// TwinCAT 3 PLC project StetigerPID_Regler
// ProgramVersion: 3.1.4022.1
// libraries:
//   Tc2_ControllerToolbox, * (Beckhoff Automation GmbH)
//   Tc2_Standard, * (Beckhoff Automation GmbH)
//   Tc2_System, * (Beckhoff Automation GmbH)
//   Tc2_TempController, * (Beckhoff Automation GmbH)
//   Tc2_Utilities, * (Beckhoff Automation GmbH)
//   Tc3_Module, * (Beckhoff Automation GmbH)
// project tree:
//   GVLs/ AN.TcGVL, DIO.TcGVL, dSub.TcGVL
//   / PlcTask.TcTTO
//   POUs/ MAIN.TcPOU, StetigerPID_Regler.TcPOU
// real-time tasks:
//   TASK PlcTask: cycle T#10ms, priority 20, ADS port 350
// motion (NC):
//   TASK NC-Task 1 SAF: cycle T#2ms, priority 4, ADS port 501
//   TASK NC-Task 1 SVB: cycle T#10ms, priority 8, ADS port 511
//   AXIS Axis 1 (id 1)
//     OtherSettings: AllowMotionCmdToSlave=true
//     encoder EncType=4
//       EncPara: MaxCount=#x0000ffff
//         Inc: RefSoftSyncMask=#x0000ffff
//     drive DrvType=24
//       Analog: ScaleFactorActTorque=0.1
//       TimeComp: TaskDelayCycles=1
//     controller CtrType=1
//       CtrPara: PriorControlFactor=1
//         Observer: BandWidth=20
//   AXIS Axis 2 (id 2)
//     OtherSettings: AllowMotionCmdToSlave=true
//     encoder EncType=4
//       EncPara: MaxCount=#x0000ffff
//         Inc: RefSoftSyncMask=#x0000ffff
//     drive DrvType=24
//       Analog: ScaleFactorActTorque=0.1
//       TimeComp: TaskDelayCycles=1
//     controller CtrType=1
//       CtrPara: PriorControlFactor=1
//         Observer: BandWidth=20
//   AXIS Axis 3 (id 3)
//     OtherSettings: AllowMotionCmdToSlave=true
//     encoder EncType=4
//       EncPara: MaxCount=#x0000ffff
//     drive DrvType=23
//       Analog: ScaleFactorActTorque=0.1
//       TimeComp: TaskDelayCycles=1
//     controller CtrType=1
//       CtrPara: PriorControlFactor=1
//         Observer: BandWidth=20
//   AXIS Axis 4 (id 4)
//     OtherSettings: AllowMotionCmdToSlave=true
//     encoder EncType=4
//       EncPara: MaxCount=#x0000ffff
//     drive DrvType=23
//       Analog: ScaleFactorActTorque=0.1
//       TimeComp: TaskDelayCycles=1
//     controller CtrType=1
//       CtrPara: PriorControlFactor=1
//         Observer: BandWidth=20
//   AXIS Axis 5 (id 5)
//     OtherSettings: AllowMotionCmdToSlave=true
//     encoder EncType=19
//       EncPara: MaxCount=#xffffffff
//     drive DrvType=16
//       DrvPara: MaxCount=#xffffffff
//         Analog: ScaleFactorActTorque=0.1
//         TimeComp: TaskDelayCycles=1
//     controller CtrType=1
//       CtrPara: PriorControlFactor=1
//         Observer: BandWidth=20
//   AXIS Axis 6 (id 6)
//     OtherSettings: AllowMotionCmdToSlave=true
//     encoder EncType=19
//       EncPara: MaxCount=#xffffffff
//     drive DrvType=16
//       DrvPara: MaxCount=#xffffffff
//         Analog: ScaleFactorActTorque=0.1
//         TimeComp: TaskDelayCycles=1
//     controller CtrType=1
//       CtrPara: PriorControlFactor=1
//         Observer: BandWidth=20
// I/O:
//   DEVICE Device 1 (EtherCAT), AmsNetId 5.35.139.20.2.1
//     Term 1 (EK1200) [EK1200-5000 EtherCAT Power supply (2A E-Bus)]
//       Term 2 (EL1809) [EL1809 16Ch. Dig. Input 24V, 3ms]
//       Term 3 (EL1809) [EL1809 16Ch. Dig. Input 24V, 3ms]
//       Term 4 (EL2809) [EL2809 16Ch. Dig. Output 24V, 0.5A]
//       Term 5 (EL2809) [EL2809 16Ch. Dig. Output 24V, 0.5A]
//       Term 6 (EL3064) [EL3064 4Ch. Ana. Input 0-10V]
//       Term 7 (EL4034) [EL4034 4Ch. Ana. Output +/-10V, 12bit]
//       Term 8 (EL7031) [EL7031 1Ch. Stepper motor output stage (24V, 1.5A)]
//       Term 9 (EL7031) [EL7031 1Ch. Stepper motor output stage (24V, 1.5A)]
//       Term 10 (EL7332) [EL7332 2Ch. DC motor output stage (24V, 1.5A)]
//       Term 11 (EL7201-0010) [EL7201-0010 1Ch. MDP742 Servo motor output stage with OCT (50V, 4A)]
//       Term 12 (EL7201-0010) [EL7201-0010 1Ch. MDP742 Servo motor output stage with OCT (50V, 4A)]
//       Term 26 (EL6090) [EL6090 Display terminal]
//       Term 27 (EK1110) [EK1110 EtherCAT extension]
// variable links:
//   NC-Task 1 SAF/Axes/Axis 1 <-> Device 1 (EtherCAT)/Term 1 (EK1200)/Term 8 (EL7031)
//     Drive/Inputs/In/nState1 @bit 3 <-> STM Status/Status/Error
//     Drive/Inputs/In/nState1 @bit 5 <-> STM Status/Status/Moving negative
//     Drive/Inputs/In/nState1 @bit 4 <-> STM Status/Status/Moving positive
//     Drive/Inputs/In/nState1 @bit 1 <-> STM Status/Status/Ready
//     Drive/Inputs/In/nState1 <-> STM Status/Status/Ready to enable
//     Drive/Inputs/In/nState1 @bit 6 <-> STM Status/Status/Torque reduced
//     Drive/Inputs/In/nState1 @bit 2 <-> STM Status/Status/Warning
//     Drive/Inputs/In/nState2 @bit 3 <-> STM Status/Status/Digital input 1
//     Drive/Inputs/In/nState2 @bit 4 <-> STM Status/Status/Digital input 2
//     Drive/Inputs/In/nState2 @bit 5 <-> STM Status/Status/Sync error
//     Drive/Inputs/In/nState2 @bit 7 <-> STM Status/Status/TxPDO Toggle
//     Drive/Inputs/In/nState4 @bit 1 <-> WcState/InputToggle
//     Drive/Inputs/In/nState4 <-> WcState/WcState
//     Drive/Outputs/Out/nCtrl1 <-> STM Control/Control/Enable
//     Drive/Outputs/Out/nCtrl1 @bit 2 <-> STM Control/Control/Reduce torque
//     Drive/Outputs/Out/nCtrl1 @bit 1 <-> STM Control/Control/Reset
//     Drive/Outputs/Out/nDataOut2[0] <-> STM Velocity/Velocity
//     Enc/Inputs/In/nDataIn1[0] <-> ENC Status compact/Counter value
//     Enc/Inputs/In/nDataIn2[0] <-> ENC Status compact/Latch value
//     Enc/Inputs/In/nState1 @bit 4 <-> ENC Status compact/Status/Counter overflow
//     Enc/Inputs/In/nState1 @bit 3 <-> ENC Status compact/Status/Counter underflow
//     Enc/Inputs/In/nState1 @bit 1 <-> ENC Status compact/Status/Latch extern valid
//     Enc/Inputs/In/nState1 @bit 2 <-> ENC Status compact/Status/Set counter done
//     Enc/Inputs/In/nState2 @bit 4 <-> ENC Status compact/Status/Status of extern latch
//     Enc/Inputs/In/nState2 @bit 5 <-> ENC Status compact/Status/Sync error
//     Enc/Inputs/In/nState2 @bit 7 <-> ENC Status compact/Status/TxPDO Toggle
//     Enc/Inputs/In/nState4 @bit 1 <-> WcState/InputToggle
//     Enc/Inputs/In/nState4 <-> WcState/WcState
//     Enc/Outputs/Out/nCtrl1 @bit 3 <-> ENC Control compact/Control/Enable latch extern on negative edge
//     Enc/Outputs/Out/nCtrl1 @bit 1 <-> ENC Control compact/Control/Enable latch extern on positive edge
//     Enc/Outputs/Out/nCtrl1 @bit 2 <-> ENC Control compact/Control/Set counter
//     Enc/Outputs/Out/nDataOut1[0] <-> ENC Control compact/Set counter value
//   NC-Task 1 SAF/Axes/Axis 2 <-> Device 1 (EtherCAT)/Term 1 (EK1200)/Term 9 (EL7031)
//     Drive/Inputs/In/nState1 @bit 3 <-> STM Status/Status/Error
//     Drive/Inputs/In/nState1 @bit 5 <-> STM Status/Status/Moving negative
//     Drive/Inputs/In/nState1 @bit 4 <-> STM Status/Status/Moving positive
//     Drive/Inputs/In/nState1 @bit 1 <-> STM Status/Status/Ready
//     Drive/Inputs/In/nState1 <-> STM Status/Status/Ready to enable
//     Drive/Inputs/In/nState1 @bit 6 <-> STM Status/Status/Torque reduced
//     Drive/Inputs/In/nState1 @bit 2 <-> STM Status/Status/Warning
//     Drive/Inputs/In/nState2 @bit 3 <-> STM Status/Status/Digital input 1
//     Drive/Inputs/In/nState2 @bit 4 <-> STM Status/Status/Digital input 2
//     Drive/Inputs/In/nState2 @bit 5 <-> STM Status/Status/Sync error
//     Drive/Inputs/In/nState2 @bit 7 <-> STM Status/Status/TxPDO Toggle
//     Drive/Inputs/In/nState4 @bit 1 <-> WcState/InputToggle
//     Drive/Inputs/In/nState4 <-> WcState/WcState
//     Drive/Outputs/Out/nCtrl1 <-> STM Control/Control/Enable
//     Drive/Outputs/Out/nCtrl1 @bit 2 <-> STM Control/Control/Reduce torque
//     Drive/Outputs/Out/nCtrl1 @bit 1 <-> STM Control/Control/Reset
//     Drive/Outputs/Out/nDataOut2[0] <-> STM Velocity/Velocity
//     Enc/Inputs/In/nDataIn1[0] <-> ENC Status compact/Counter value
//     Enc/Inputs/In/nDataIn2[0] <-> ENC Status compact/Latch value
//     Enc/Inputs/In/nState1 @bit 4 <-> ENC Status compact/Status/Counter overflow
//     Enc/Inputs/In/nState1 @bit 3 <-> ENC Status compact/Status/Counter underflow
//     Enc/Inputs/In/nState1 @bit 1 <-> ENC Status compact/Status/Latch extern valid
//     Enc/Inputs/In/nState1 @bit 2 <-> ENC Status compact/Status/Set counter done
//     Enc/Inputs/In/nState2 @bit 4 <-> ENC Status compact/Status/Status of extern latch
//     Enc/Inputs/In/nState2 @bit 5 <-> ENC Status compact/Status/Sync error
//     Enc/Inputs/In/nState2 @bit 7 <-> ENC Status compact/Status/TxPDO Toggle
//     Enc/Inputs/In/nState4 @bit 1 <-> WcState/InputToggle
//     Enc/Inputs/In/nState4 <-> WcState/WcState
//     Enc/Outputs/Out/nCtrl1 @bit 3 <-> ENC Control compact/Control/Enable latch extern on negative edge
//     Enc/Outputs/Out/nCtrl1 @bit 1 <-> ENC Control compact/Control/Enable latch extern on positive edge
//     Enc/Outputs/Out/nCtrl1 @bit 2 <-> ENC Control compact/Control/Set counter
//     Enc/Outputs/Out/nDataOut1[0] <-> ENC Control compact/Set counter value
//   NC-Task 1 SAF/Axes/Axis 3 <-> Device 1 (EtherCAT)/Term 1 (EK1200)/Term 10 (EL7332)
//     Drive/Inputs/In/nState1 @bit 3 <-> DCM Status Channel 1/Status/Error
//     Drive/Inputs/In/nState1 @bit 5 <-> DCM Status Channel 1/Status/Moving negative
//     Drive/Inputs/In/nState1 @bit 4 <-> DCM Status Channel 1/Status/Moving positive
//     Drive/Inputs/In/nState1 @bit 1 <-> DCM Status Channel 1/Status/Ready
//     Drive/Inputs/In/nState1 <-> DCM Status Channel 1/Status/Ready to enable
//     Drive/Inputs/In/nState1 @bit 6 <-> DCM Status Channel 1/Status/Torque reduced
//     Drive/Inputs/In/nState1 @bit 2 <-> DCM Status Channel 1/Status/Warning
//     Drive/Inputs/In/nState2 @bit 3 <-> DCM Status Channel 1/Status/Digital input 1
//     Drive/Inputs/In/nState2 @bit 4 <-> DCM Status Channel 1/Status/Digital input 2
//     Drive/Inputs/In/nState2 @bit 5 <-> DCM Status Channel 1/Status/Sync error
//     Drive/Inputs/In/nState2 @bit 7 <-> DCM Status Channel 1/Status/TxPDO Toggle
//     Drive/Inputs/In/nState4 @bit 1 <-> WcState/InputToggle
//     Drive/Inputs/In/nState4 <-> WcState/WcState
//     Drive/Outputs/Out/nCtrl1 <-> DCM Control Channel 1/Control/Enable
//     Drive/Outputs/Out/nCtrl1 @bit 2 <-> DCM Control Channel 1/Control/Reduce torque
//     Drive/Outputs/Out/nCtrl1 @bit 1 <-> DCM Control Channel 1/Control/Reset
//     Drive/Outputs/Out/nDataOut2[0] <-> DCM Velocity Channel 1/Velocity
//   NC-Task 1 SAF/Axes/Axis 4 <-> Device 1 (EtherCAT)/Term 1 (EK1200)/Term 10 (EL7332)
//     Drive/Inputs/In/nState1 @bit 3 <-> DCM Status Channel 2/Status/Error
//     Drive/Inputs/In/nState1 @bit 5 <-> DCM Status Channel 2/Status/Moving negative
//     Drive/Inputs/In/nState1 @bit 4 <-> DCM Status Channel 2/Status/Moving positive
//     Drive/Inputs/In/nState1 @bit 1 <-> DCM Status Channel 2/Status/Ready
//     Drive/Inputs/In/nState1 <-> DCM Status Channel 2/Status/Ready to enable
//     Drive/Inputs/In/nState1 @bit 6 <-> DCM Status Channel 2/Status/Torque reduced
//     Drive/Inputs/In/nState1 @bit 2 <-> DCM Status Channel 2/Status/Warning
//     Drive/Inputs/In/nState2 @bit 3 <-> DCM Status Channel 2/Status/Digital input 1
//     Drive/Inputs/In/nState2 @bit 4 <-> DCM Status Channel 2/Status/Digital input 2
//     Drive/Inputs/In/nState2 @bit 5 <-> DCM Status Channel 2/Status/Sync error
//     Drive/Inputs/In/nState2 @bit 7 <-> DCM Status Channel 2/Status/TxPDO Toggle
//     Drive/Inputs/In/nState4 @bit 1 <-> WcState/InputToggle
//     Drive/Inputs/In/nState4 <-> WcState/WcState
//     Drive/Outputs/Out/nCtrl1 <-> DCM Control Channel 2/Control/Enable
//     Drive/Outputs/Out/nCtrl1 @bit 2 <-> DCM Control Channel 2/Control/Reduce torque
//     Drive/Outputs/Out/nCtrl1 @bit 1 <-> DCM Control Channel 2/Control/Reset
//     Drive/Outputs/Out/nDataOut2[0] <-> DCM Velocity Channel 2/Velocity
//   NC-Task 1 SAF/Axes/Axis 5 <-> Device 1 (EtherCAT)/Term 1 (EK1200)/Term 11 (EL7201-0010)
//     Drive/Inputs/In/nDcOutputTime <-> InfoData/DcOutputShift
//     Drive/Inputs/In/nState1 <-> DRV Statusword/Statusword
//     Drive/Inputs/In/nState2 <-> DRV Statusword/Statusword @bit 8
//     Drive/Inputs/In/nState4 @bit 1 <-> WcState/InputToggle
//     Drive/Inputs/In/nState4 <-> WcState/WcState
//     Drive/Outputs/Out/nCtrl1 <-> DRV Controlword/Controlword
//     Drive/Outputs/Out/nCtrl2 <-> DRV Controlword/Controlword @bit 8
//     Drive/Outputs/Out/nDataOut2 <-> DRV Target velocity/Target velocity
//     Enc/Inputs/In/nDataIn1 <-> FB Position/Position
//     Enc/Inputs/In/nDcInputTime <-> InfoData/DcInputShift
//     Enc/Inputs/In/nState4 @bit 1 <-> WcState/InputToggle
//     Enc/Inputs/In/nState4 <-> WcState/WcState
//   NC-Task 1 SAF/Axes/Axis 6 <-> Device 1 (EtherCAT)/Term 1 (EK1200)/Term 12 (EL7201-0010)
//     Drive/Inputs/In/nDcOutputTime <-> InfoData/DcOutputShift
//     Drive/Inputs/In/nState1 <-> DRV Statusword/Statusword
//     Drive/Inputs/In/nState2 <-> DRV Statusword/Statusword @bit 8
//     Drive/Inputs/In/nState4 @bit 1 <-> WcState/InputToggle
//     Drive/Inputs/In/nState4 <-> WcState/WcState
//     Drive/Outputs/Out/nCtrl1 <-> DRV Controlword/Controlword
//     Drive/Outputs/Out/nCtrl2 <-> DRV Controlword/Controlword @bit 8
//     Drive/Outputs/Out/nDataOut2 <-> DRV Target velocity/Target velocity
//     Enc/Inputs/In/nDataIn1 <-> FB Position/Position
//     Enc/Inputs/In/nDcInputTime <-> InfoData/DcInputShift
//     Enc/Inputs/In/nState4 @bit 1 <-> WcState/InputToggle
//     Enc/Inputs/In/nState4 <-> WcState/WcState
//   StetigerPID_Regler/StetigerPID_Regler Instance <-> Device 1 (EtherCAT)/Term 1 (EK1200)/Term 2 (EL1809)
//     PlcTask Inputs/dSub.B1 <-> Channel 1/Input
//     PlcTask Inputs/dSub.B2 <-> Channel 2/Input
//     PlcTask Inputs/dSub.S1 <-> Channel 4/Input
//     PlcTask Inputs/dSub.S10 <-> Channel 12/Input
//     PlcTask Inputs/dSub.S11 <-> Channel 13/Input
//     PlcTask Inputs/dSub.S2 <-> Channel 3/Input
//     PlcTask Inputs/dSub.S3 <-> Channel 6/Input
//     PlcTask Inputs/dSub.S4 <-> Channel 5/Input
//     PlcTask Inputs/dSub.S5 <-> Channel 8/Input
//     PlcTask Inputs/dSub.S6 <-> Channel 7/Input
//     PlcTask Inputs/dSub.S7 <-> Channel 10/Input
//     PlcTask Inputs/dSub.S8 <-> Channel 9/Input
//     PlcTask Inputs/dSub.S9 <-> Channel 11/Input
//   StetigerPID_Regler/StetigerPID_Regler Instance <-> Device 1 (EtherCAT)/Term 1 (EK1200)/Term 3 (EL1809)
//     PlcTask Inputs/DIO.DI_{1..16} <-> Channel {1..16}/Input  (16 links)
//   StetigerPID_Regler/StetigerPID_Regler Instance <-> Device 1 (EtherCAT)/Term 1 (EK1200)/Term 4 (EL2809)
//     PlcTask Outputs/dSub.P{1..4} <-> Channel {3..6}/Output  (4 links)
//     PlcTask Outputs/dSub.Q1 <-> Channel 1/Output
//     PlcTask Outputs/dSub.Q2 <-> Channel 2/Output
//   StetigerPID_Regler/StetigerPID_Regler Instance <-> Device 1 (EtherCAT)/Term 1 (EK1200)/Term 5 (EL2809)
//     PlcTask Outputs/DIO.DQ_{1..16} <-> Channel {1..16}/Output  (16 links)
//   StetigerPID_Regler/StetigerPID_Regler Instance <-> Device 1 (EtherCAT)/Term 1 (EK1200)/Term 6 (EL3064)
//     PlcTask Inputs/AN.AI_1 <-> AI Standard Channel 3/Value
//     PlcTask Inputs/AN.AI_2 <-> AI Standard Channel 4/Value
//     PlcTask Inputs/dSub.AI_0 <-> AI Standard Channel 1/Value
//     PlcTask Inputs/dSub.AI_1 <-> AI Standard Channel 2/Value
//   StetigerPID_Regler/StetigerPID_Regler Instance <-> Device 1 (EtherCAT)/Term 1 (EK1200)/Term 7 (EL4034)
//     PlcTask Outputs/AN.AQ_1 <-> AO Outputs Channel 3/Analog output
//     PlcTask Outputs/AN.AQ_2 <-> AO Outputs Channel 4/Analog output
//     PlcTask Outputs/dSub.AQ_0 <-> AO Outputs Channel 1/Analog output

CONFIGURATION StetigerPID_Regler
    RESOURCE PLC ON TwinCAT3
        TASK PlcTask(INTERVAL := T#10ms, PRIORITY := 20);
        PROGRAM MAIN WITH PlcTask : MAIN;
    END_RESOURCE
END_CONFIGURATION

// ---- GVLs/AN.TcGVL
{attribute 'qualified_only'}
VAR_GLOBAL
	// Analogeingang AI 1	
	AI_1 AT %I*: INT;
 	// Analogeingang AI 2	
	AI_2 AT %I*: INT;
	// Analogausgang AQ 1	
	AQ_1 AT %Q*: INT;
 	// Analogausgang AQ 2	
	AQ_2 AT %Q*: INT;
END_VAR

// ---- GVLs/DIO.TcGVL
{attribute 'qualified_only'}
VAR_GLOBAL
	// Digitaler Eingang 1
	DI_1 AT %I*: BOOL; 
	// Digitaler Eingang 2
	DI_2 AT %I*: BOOL; 	
	// Digitaler Eingang 3
	DI_3 AT %I*: BOOL; 
	// Digitaler Eingang 4
	DI_4 AT %I*: BOOL; 		
	// Digitaler Eingang 5
	DI_5 AT %I*: BOOL; 
	// Digitaler Eingang 6
	DI_6 AT %I*: BOOL; 	
	// Digitaler Eingang 7
	DI_7 AT %I*: BOOL; 
	// Digitaler Eingang 8
	DI_8 AT %I*: BOOL; 
	// Digitaler Eingang 9
	DI_9 AT %I*: BOOL; 
	// Digitaler Eingang 10
	DI_10 AT %I*: BOOL; 	
	// Digitaler Eingang 11
	DI_11 AT %I*: BOOL; 
	// Digitaler Eingang 12
	DI_12 AT %I*: BOOL; 		
	// Digitaler Eingang 13
	DI_13 AT %I*: BOOL; 
	// Digitaler Eingang 14
	DI_14 AT %I*: BOOL; 	
	// Digitaler Eingang 15
	DI_15 AT %I*: BOOL; 
	// Digitaler Eingang 16
	DI_16 AT %I*: BOOL; 
	
	// Digitaler Ausgang 1
	DQ_1 AT %Q*: BOOL; 
	// Digitaler Ausgang 2
	DQ_2 AT %Q*: BOOL; 	
	// Digitaler Ausgang 3
	DQ_3 AT %Q*: BOOL; 
	// Digitaler Ausgang 4
	DQ_4 AT %Q*: BOOL; 		
	// Digitaler Ausgang 5
	DQ_5 AT %Q*: BOOL; 
	// Digitaler Ausgang 6
	DQ_6 AT %Q*: BOOL; 	
	// Digitaler Ausgang 7
	DQ_7 AT %Q*: BOOL; 
	// Digitaler Ausgang 8
	DQ_8 AT %Q*: BOOL; 
	// Digitaler Ausgang 9
	DQ_9 AT %Q*: BOOL; 
	// Digitaler Ausgang 10
	DQ_10 AT %Q*: BOOL; 	
	// Digitaler Ausgang 11
	DQ_11 AT %Q*: BOOL; 
	// Digitaler Ausgang 12
	DQ_12 AT %Q*: BOOL; 		
	// Digitaler Ausgang 13
	DQ_13 AT %Q*: BOOL; 
	// Digitaler Ausgang 14
	DQ_14 AT %Q*: BOOL; 	
	// Digitaler Ausgang 15
	DQ_15 AT %Q*: BOOL; 
	// Digitaler Ausgang 16
	DQ_16 AT %Q*: BOOL; 	
END_VAR

// ---- GVLs/dSub.TcGVL
{attribute 'qualified_only'}
VAR_GLOBAL
	
	// Linearantrieb Endlage links (Öffner)
	B1 AT %I*: BOOL; 
	// Linearantrieb Endlage rechts (Öffner)
	B2 AT %I*: BOOL;
	// Taster (1) (Schliesser)
	S1 AT %I*: BOOL;	
	// Taster (0) (Öffner)
	S2 AT %I*: BOOL;
	// Taster I (Schliesser)
	S3 AT %I*: BOOL;
	// Taster II (Schliesser)
	S4 AT %I*: BOOL;
	// Taster Pfeil auf (Schliesser)
	S5 AT %I*: BOOL;
	// Taster Pfeil ab (Schliesser)
	S6 AT %I*: BOOL;
	// Taster + (Schliesser)
	S7 AT %I*: BOOL;
	// Taster - (Schliesser)
	S8 AT %I*: BOOL;
	// Taster STOP (Öffner)
	S9 AT %I*: BOOL;
	// Taster Not Halt (Öffner)
	S10 AT %I*: BOOL;
	// Taster Not Halt (Schliesser)
	S11 AT %I*: BOOL;
	
	// Analogeingang 0
	AI_0 AT %I*: INT;
	// Analogeingang 1
	AI_1 AT %I*: INT;	
	
	// Linearantrieb Rechtslauf
	Q1 AT %Q*: BOOL;
	// Linearantrieb Linkslauf
	Q2 AT %Q*: BOOL;
	// Meldeleuchte im Taster S1 (weiß)
	P1 AT %Q*: BOOL;
	// Meldeleuchte weiß
	P2 AT %Q*: BOOL;
	// Meldeleuchte rot
	P3 AT %Q*: BOOL;
	// Meldeleuchte grün
	P4 AT %Q*: BOOL;

	// Analogausgang 0
	AQ_0 AT %Q*: INT;
	
END_VAR

// ---- POUs/MAIN.TcPOU
PROGRAM MAIN
VAR

END_VAR

StetigerPID_Regler();

END_PROGRAM

// ---- POUs/StetigerPID_Regler.TcPOU
PROGRAM StetigerPID_Regler
VAR
	fSetpointValue					: FLOAT		:= 5.0;
	fActualValue					: FLOAT;
	fManSyncValue				: FLOAT;
	bSync							: BOOL;

	fOut							: FLOAT;
	bHold							: BOOL;

	eMode							: E_CTRL_MODE;
	stCTRL_PID_PARAMS		: ST_CTRL_PID_PARAMS;

	eErrorId						: E_CTRL_ERRORCODES;
	bError							: BOOL;
	bARWactive					: BOOL;

	(* controller *)
	fbCTRL_PID					: FB_CTRL_PID;

	bInit							: BOOL	:= TRUE;
	fbTON							: TON;
	
	fSetpointValueToScope: LREAL;
	fActualValueToScope: LREAL;
	fOutToScope: LREAL;
END_VAR



IF bInit
THEN
	(* init parameter struct *)
	stCTRL_PID_PARAMS.tCtrlCycleTime		:= T#10ms;
	stCTRL_PID_PARAMS.tTaskCycleTime		:= T#10ms;
	stCTRL_PID_PARAMS.fKp					:= 2.0;			(* proportional gain Kp				*)
	stCTRL_PID_PARAMS.tTn					:= T#1s;		(*  Tn									*)
	stCTRL_PID_PARAMS.tTv					:= T#200ms;	(*  Tv									*)
	stCTRL_PID_PARAMS.tTd					:= T#100ms;	(*  Td									*)
	stCTRL_PID_PARAMS.fOutMaxLimit			:=  32765;			(* maximum output limit				*)
	stCTRL_PID_PARAMS.fOutMinLimit			:= 0;			(* minimum output limit				*)

	(* set the mode to ACTIVE --> normal operation *)
	eMode							:= eCTRL_MODE_ACTIVE;

	(* reset the init flag *)
	bInit							:= FALSE;
END_IF

fSetpointValue := 2000;

		fActualValue := AN.AI_1;
		fActualValue := fActualValue / 8.18;


(* copy var to scope var *)
fSetpointValueToScope 	:= fSetpointValue;
fActualValueToScope 		:= fActualValue;


(* call controller *)
fbCTRL_PID(		fSetpointValue		:= fSetpointValue,
					fActualValue		:= fActualValue,
					fManSyncValue	:= fManSyncValue,
					bSync				:= bSync,
					eMode				:= eMode,
					bHold				:= bHold,
					stParams			:= stCTRL_PID_PARAMS,
					fOut				=> fOut,
					bARWactive		=> bARWactive,
					eErrorId			=> eErrorId,
					bError				=> bError
				);


(* copy var to scope var *)

fOutToScope := fOut;
AN.AQ_1 :=  LREAL_TO_UINT (fOut);

END_PROGRAM
